// Tests exercise the public input/output and command contracts.
FUNCTION_BLOCK FB_TwoPosActuator_Test EXTENDS TcUnit.FB_TestSuite

InitialStateIsUndefined();
UndefinedBecomesAdvancedOnFeedback();
UndefinedBecomesRetractedOnFeedback();
UndefinedFaultsWhenBothFeedbacksAssertSimultaneously();
AdvanceCommandDrivesStateToAdvancing();
AdvanceAtPositionRearms();
AdvanceRejectedWhenPermissiveNotMet();
AdvanceRejectedFromOperatorWhileSourceLocked();
AdvancingCompletesOnAdvancedFeedback();
AdvancingFaultsOnBothFeedback();
AdvancedFaultsOnLostFeedback();
RetractFromAdvancedDrivesRetracting();
AbortAlwaysAcceptedAndReturnsToUndefined();
ResetClearsFaultAndReturnsToUndefined();
HeaderBusyMirrorsMovingState();

METHOD InitialStateIsUndefined
VAR
    fb : TcForge.FB_TwoPosActuator;
END_VAR
TEST('InitialStateIsUndefined');

// No feedbacks, one cycle. currentState init is Undefined and the body
// only transitions out when a single feedback asserts.
fb();

AssertEquals_DINT(
    Expected := TcForge.E_TwoPosActuator_State.Undefined,
    Actual   := fb.sts.state,
    Message  := 'Fresh instance with no feedbacks must stay in Undefined');
AssertFalse(
    Condition := fb.outAdvance,
    Message   := 'Undefined state must de-energize outValveAdvance');
AssertFalse(
    Condition := fb.outRetract,
    Message   := 'Undefined state must de-energize outValveRetract');
AssertFalse(
    Condition := fb.sts.header.faulted,
    Message   := 'Fresh instance must not be faulted');

TEST_FINISHED();
END_METHOD

METHOD UndefinedBecomesAdvancedOnFeedback
VAR
    fb : TcForge.FB_TwoPosActuator;
END_VAR
TEST('UndefinedBecomesAdvancedOnFeedback');

// Simulate a device that was already at the advanced end-stop on boot.
fb.inAdvanced := TRUE;
fb();

AssertEquals_DINT(
    Expected := TcForge.E_TwoPosActuator_State.Advanced,
    Actual   := fb.sts.state,
    Message  := 'Undefined must latch to Advanced when only inFbkAdvanced is TRUE');
AssertTrue(
    Condition := fb.sts.advanced,
    Message   := 'advanced must follow the resolved state');
AssertFalse(
    Condition := fb.sts.retracted,
    Message   := 'retracted must be FALSE when Advanced');

TEST_FINISHED();
END_METHOD

METHOD UndefinedBecomesRetractedOnFeedback
VAR
    fb : TcForge.FB_TwoPosActuator;
END_VAR
TEST('UndefinedBecomesRetractedOnFeedback');

fb.inRetracted := TRUE;
fb();

AssertEquals_DINT(
    Expected := TcForge.E_TwoPosActuator_State.Retracted,
    Actual   := fb.sts.state,
    Message  := 'Undefined must latch to Retracted when only inFbkRetracted is TRUE');
AssertTrue(
    Condition := fb.sts.retracted,
    Message   := 'retracted must follow the resolved state');
AssertFalse(
    Condition := fb.sts.advanced,
    Message   := 'advanced must be FALSE when Retracted');

TEST_FINISHED();
END_METHOD

METHOD UndefinedFaultsWhenBothFeedbacksAssertSimultaneously
VAR
    fb : TcForge.FB_TwoPosActuator;
END_VAR
TEST('UndefinedFaultsWhenBothFeedbacksAssertSimultaneously');

// A physically impossible sensor state — both end-stops asserted. The FB
// must trip to Fault with BothFeedbackOn instead of silently picking
// one branch.
fb.inAdvanced := TRUE;
fb.inRetracted := TRUE;
fb();

AssertEquals_DINT(
    Expected := TcForge.E_TwoPosActuator_State.Fault,
    Actual   := fb.sts.state,
    Message  := 'Both feedbacks simultaneously must drive state to Fault');
AssertTrue(
    Condition := fb.sts.header.faulted,
    Message   := 'header must report faulted when both feedbacks assert');
AssertEquals_DINT(
    Expected := TcForge.E_TwoPosActuator_Fault.BothFeedbackOn,
    Actual   := fb.sts.header.faultCode,
    Message  := 'Active fault code must be BothFeedbackOn');
AssertFalse(
    Condition := fb.outAdvance,
    Message   := 'Fault state must de-energize outValveAdvance');
AssertFalse(
    Condition := fb.outRetract,
    Message   := 'Fault state must de-energize outValveRetract');

TEST_FINISHED();
END_METHOD

METHOD AdvanceCommandDrivesStateToAdvancing
VAR
    fb   : TcForge.FB_TwoPosActuator;
    resp : TcForge.E_RpcMethodResponse;
END_VAR
TEST('AdvanceCommandDrivesStateToAdvancing');

// Start from Retracted (single known end-stop) — the canonical starting
// point before an Advance command.
fb.inRetracted := TRUE;
fb();
AssertEquals_DINT(
    Expected := TcForge.E_TwoPosActuator_State.Retracted,
    Actual   := fb.sts.state,
    Message  := 'Precondition: feedback-only start must settle to Retracted');

// Drop the retracted feedback first (simulates real physical travel) so
// the Advancing branch isn't racing against a lost-feedback trip.
fb.inRetracted := FALSE;

resp := fb.Advance(eRequester := TcForge.E_Requester.PROG);
fb();

AssertEquals_DINT(
    Expected := TcForge.E_RpcMethodResponse.ACCEPTED,
    Actual   := resp,
    Message  := 'Advance from PROG in Retracted must be ACCEPTED');
AssertEquals_DINT(
    Expected := TcForge.E_TwoPosActuator_State.Advancing,
    Actual   := fb.sts.state,
    Message  := 'Accepted Advance must transition state to Advancing');
AssertTrue(
    Condition := fb.outAdvance,
    Message   := 'Advancing state must energize outValveAdvance');
AssertFalse(
    Condition := fb.outRetract,
    Message   := 'Advancing state must NOT energize outValveRetract');
AssertTrue(
    Condition := fb.sts.moving,
    Message   := 'moving must flag the Advancing transit');

TEST_FINISHED();
END_METHOD

METHOD AdvanceAtPositionRearms
VAR
    fb   : TcForge.FB_TwoPosActuator;
    resp : TcForge.E_RpcMethodResponse;
END_VAR
TEST('AdvanceAtPositionRearms');

fb.inAdvanced := TRUE;
fb();
AssertEquals_DINT(
    Expected := TcForge.E_TwoPosActuator_State.Advanced,
    Actual   := fb.sts.state,
    Message  := 'Precondition: must be Advanced before rearming');

resp := fb.Advance(eRequester := TcForge.E_Requester.PROG);

AssertEquals_DINT(
    Expected := TcForge.E_RpcMethodResponse.ACCEPTED,
    Actual   := resp,
    Message  := 'Advance at known position explicitly rearms the device');

TEST_FINISHED();
END_METHOD

METHOD AdvanceRejectedWhenPermissiveNotMet
VAR
    fb   : TcForge.FB_TwoPosActuator;
    resp : TcForge.E_RpcMethodResponse;
END_VAR
TEST('AdvanceRejectedWhenPermissiveNotMet');

// Force the advance permissive to fail. One cycle is enough to let
// advancePermissives refresh sts.bOK to FALSE before we call Advance.
fb.MapAdvanceCondition(bitIndex := 0, bGood := FALSE);
fb();
fb.inRetracted := FALSE;

resp := fb.Advance(eRequester := TcForge.E_Requester.PROG);

AssertEquals_DINT(
    Expected := TcForge.E_RpcMethodResponse.REJECTED_PERMISSIVE_NOT_MET,
    Actual   := resp,
    Message  := 'Advance must be rejected when advancePermissives.sts.bOK is FALSE');

TEST_FINISHED();
END_METHOD

METHOD AdvanceRejectedFromOperatorWhileSourceLocked
VAR
    fb   : TcForge.FB_TwoPosActuator;
    resp : TcForge.E_RpcMethodResponse;
END_VAR
TEST('AdvanceRejectedFromOperatorWhileSourceLocked');

fb.LockSource(bLock := TRUE);
resp := fb.Advance(eRequester := TcForge.E_Requester.OPERATOR);

AssertEquals_DINT(
    Expected := TcForge.E_RpcMethodResponse.REJECTED_SOURCE_NOT_ALLOWED,
    Actual   := resp,
    Message  := 'OPERATOR must be rejected while source-locked');

TEST_FINISHED();
END_METHOD

METHOD AdvancingCompletesOnAdvancedFeedback
VAR
    fb : TcForge.FB_TwoPosActuator;
END_VAR
TEST('AdvancingCompletesOnAdvancedFeedback');

// One warmup cycle so advancePermissives refreshes sts.bOK to TRUE
// (unmapped bits default good). Without it the cached bOK is still
// FALSE on a fresh instance and Advance() gets rejected with
// REJECTED_PERMISSIVE_NOT_MET.
fb();
fb.Advance(eRequester := TcForge.E_Requester.PROG);
fb();
AssertEquals_DINT(
    Expected := TcForge.E_TwoPosActuator_State.Advancing,
    Actual   := fb.sts.state,
    Message  := 'Precondition: must be in Advancing');

fb.inAdvanced := TRUE;
fb();

AssertEquals_DINT(
    Expected := TcForge.E_TwoPosActuator_State.Advanced,
    Actual   := fb.sts.state,
    Message  := 'Advancing must complete to Advanced when inFbkAdvanced asserts');
AssertFalse(
    Condition := fb.sts.moving,
    Message   := 'moving must clear once the motion completes');

TEST_FINISHED();
END_METHOD

METHOD AdvancingFaultsOnBothFeedback
VAR
    fb : TcForge.FB_TwoPosActuator;
END_VAR
TEST('AdvancingFaultsOnBothFeedback');

// Warmup cycle so advancePermissives reports bOK before Advance().
fb();
fb.Advance(eRequester := TcForge.E_Requester.PROG);
fb();

// Simulate a stuck or failed retracted end-stop latching HIGH while the
// actuator is already reporting Advanced — classic dual-sensor fault.
fb.inAdvanced := TRUE;
fb.inRetracted := TRUE;
fb();

AssertEquals_DINT(
    Expected := TcForge.E_TwoPosActuator_State.Fault,
    Actual   := fb.sts.state,
    Message  := 'Both feedbacks while Advancing must trip to Fault');
AssertEquals_DINT(
    Expected := TcForge.E_TwoPosActuator_Fault.BothFeedbackOn,
    Actual   := fb.sts.header.faultCode,
    Message  := 'Fault code must be BothFeedbackOn — the highest-priority feedback fault');

TEST_FINISHED();
END_METHOD

METHOD AdvancedFaultsOnLostFeedback
VAR
    fb : TcForge.FB_TwoPosActuator;
END_VAR
TEST('AdvancedFaultsOnLostFeedback');

fb.inAdvanced := TRUE;
fb();
AssertEquals_DINT(
    Expected := TcForge.E_TwoPosActuator_State.Advanced,
    Actual   := fb.sts.state,
    Message  := 'Precondition: must be in Advanced');

// Feedback drops while the actuator is supposed to be at the end-stop
// (wire break, loose sensor, etc.). The FB must not silently revert to
// Undefined — that would let downstream sequencing assume a known state
// that isn't actually valid.
fb.inAdvanced := FALSE;
fb();

AssertEquals_DINT(
    Expected := TcForge.E_TwoPosActuator_State.Fault,
    Actual   := fb.sts.state,
    Message  := 'Lost advanced feedback must trip to Fault, not silently revert');
AssertEquals_DINT(
    Expected := TcForge.E_TwoPosActuator_Fault.UndefinedState,
    Actual   := fb.sts.header.faultCode,
    Message  := 'Fault code must be UndefinedState when Advanced feedback disappears');

TEST_FINISHED();
END_METHOD

METHOD RetractFromAdvancedDrivesRetracting
VAR
    fb   : TcForge.FB_TwoPosActuator;
    resp : TcForge.E_RpcMethodResponse;
END_VAR
TEST('RetractFromAdvancedDrivesRetracting');

fb.inAdvanced := TRUE;
fb();
fb.inAdvanced := FALSE;

resp := fb.Retract(eRequester := TcForge.E_Requester.PROG);
fb();

AssertEquals_DINT(
    Expected := TcForge.E_RpcMethodResponse.ACCEPTED,
    Actual   := resp,
    Message  := 'Retract from Advanced must be ACCEPTED');
AssertEquals_DINT(
    Expected := TcForge.E_TwoPosActuator_State.Retracting,
    Actual   := fb.sts.state,
    Message  := 'Accepted Retract must transition to Retracting');
AssertTrue(
    Condition := fb.outRetract,
    Message   := 'Retracting must energize outValveRetract');
AssertFalse(
    Condition := fb.outAdvance,
    Message   := 'Retracting must NOT energize outValveAdvance');

TEST_FINISHED();
END_METHOD

METHOD AbortAlwaysAcceptedAndReturnsToUndefined
VAR
    fb   : TcForge.FB_TwoPosActuator;
    resp : TcForge.E_RpcMethodResponse;
END_VAR
TEST('AbortAlwaysAcceptedAndReturnsToUndefined');

// Set up a worst-case: source-locked AND in motion AND commanded by
// OPERATOR. Abort must still land. Warmup cycle first so
// advancePermissives reports bOK before Advance().
fb();
fb.LockSource(bLock := TRUE);
fb.Advance(eRequester := TcForge.E_Requester.PROG);
fb();
AssertEquals_DINT(
    Expected := TcForge.E_TwoPosActuator_State.Advancing,
    Actual   := fb.sts.state,
    Message  := 'Precondition: must be Advancing before Abort');

resp := fb.Abort(eRequester := TcForge.E_Requester.OPERATOR);
fb();

AssertEquals_DINT(
    Expected := TcForge.E_RpcMethodResponse.ACCEPTED,
    Actual   := resp,
    Message  := 'Abort must be accepted from OPERATOR even when source-locked (safety invariant)');
AssertEquals_DINT(
    Expected := TcForge.E_TwoPosActuator_State.Undefined,
    Actual   := fb.sts.state,
    Message  := 'Abort must return state to Undefined for re-evaluation');
AssertFalse(
    Condition := fb.outAdvance,
    Message   := 'Abort must de-energize outValveAdvance');
AssertFalse(
    Condition := fb.outRetract,
    Message   := 'Abort must de-energize outValveRetract');

TEST_FINISHED();
END_METHOD

METHOD ResetClearsFaultAndReturnsToUndefined
VAR
    fb   : TcForge.FB_TwoPosActuator;
    resp : TcForge.E_RpcMethodResponse;
END_VAR
TEST('ResetClearsFaultAndReturnsToUndefined');

// Trip to Fault via the both-feedbacks path.
fb.inAdvanced := TRUE;
fb.inRetracted := TRUE;
fb();
AssertTrue(
    Condition := fb.sts.header.faulted,
    Message   := 'Precondition: must be faulted before Reset');

// Drop the conflicting feedback so Reset can actually settle.
fb.inRetracted := FALSE;
fb.inAdvanced := FALSE;

resp := fb.Reset(eRequester := TcForge.E_Requester.OPERATOR);
fb();

AssertEquals_DINT(
    Expected := TcForge.E_RpcMethodResponse.ACCEPTED,
    Actual   := resp,
    Message  := 'Reset must always be accepted (safety invariant inherited from FB_DeviceBase)');
AssertFalse(
    Condition := fb.sts.header.faulted,
    Message   := 'Reset must clear the active fault');
AssertEquals_DINT(
    Expected := TcForge.E_TwoPosActuator_State.Undefined,
    Actual   := fb.sts.state,
    Message  := 'Reset must drop the state machine back to Undefined');
AssertTrue(
    Condition := fb.sts.header.lastFaultCode = TcForge.E_TwoPosActuator_Fault.BothFeedbackOn,
    Message   := 'Reset must preserve lastFaultCode for HMI post-mortem');

TEST_FINISHED();
END_METHOD

METHOD HeaderBusyMirrorsMovingState
VAR
    fb : TcForge.FB_TwoPosActuator;
END_VAR
TEST('HeaderBusyMirrorsMovingState');

// Warmup cycle so advancePermissives reports bOK before Advance().
fb();
fb.Advance(eRequester := TcForge.E_Requester.PROG);
fb();

AssertTrue(
    Condition := fb.sts.moving,
    Message   := 'Advancing must set moving');
AssertTrue(
    Condition := fb.sts.header.busy,
    Message   := 'header.busy must mirror moving so generic HMIs can show motion');
AssertFalse(
    Condition := fb.sts.header.ready,
    Message   := 'ready must be FALSE while the actuator is in motion');

TEST_FINISHED();
END_METHOD

END_FUNCTION_BLOCK

(* stored: Version 1.1.0.1, ProductVersion 3.1.4026.12
   POU FB_TwoPosActuator_Test: Id {b1c2d3e4-f5a6-7890-abcd-000000000c00}, SpecialFunc None
   Method InitialStateIsUndefined: Id {b1c2d3e4-f5a6-7890-abcd-000000000c01}
   Method UndefinedBecomesAdvancedOnFeedback: Id {b1c2d3e4-f5a6-7890-abcd-000000000c02}
   Method UndefinedBecomesRetractedOnFeedback: Id {b1c2d3e4-f5a6-7890-abcd-000000000c03}
   Method UndefinedFaultsWhenBothFeedbacksAssertSimultaneously: Id {b1c2d3e4-f5a6-7890-abcd-000000000c04}
   Method AdvanceCommandDrivesStateToAdvancing: Id {b1c2d3e4-f5a6-7890-abcd-000000000c05}
   Method AdvanceAtPositionRearms: Id {b1c2d3e4-f5a6-7890-abcd-000000000c06}
   Method AdvanceRejectedWhenPermissiveNotMet: Id {b1c2d3e4-f5a6-7890-abcd-000000000c07}
   Method AdvanceRejectedFromOperatorWhileSourceLocked: Id {b1c2d3e4-f5a6-7890-abcd-000000000c08}
   Method AdvancingCompletesOnAdvancedFeedback: Id {b1c2d3e4-f5a6-7890-abcd-000000000c09}
   Method AdvancingFaultsOnBothFeedback: Id {b1c2d3e4-f5a6-7890-abcd-000000000c0a}
   Method AdvancedFaultsOnLostFeedback: Id {b1c2d3e4-f5a6-7890-abcd-000000000c0b}
   Method RetractFromAdvancedDrivesRetracting: Id {b1c2d3e4-f5a6-7890-abcd-000000000c0c}
   Method AbortAlwaysAcceptedAndReturnsToUndefined: Id {b1c2d3e4-f5a6-7890-abcd-000000000c0d}
   Method ResetClearsFaultAndReturnsToUndefined: Id {b1c2d3e4-f5a6-7890-abcd-000000000c0e}
   Method HeaderBusyMirrorsMovingState: Id {b1c2d3e4-f5a6-7890-abcd-000000000c0f} *)
